TYPE ST_Robot_HMI :
STRUCT
	bStart : BOOL;
	bStop : BOOL;
	bInit : BOOL;
	bPowerOn : BOOL;
	bPowerOff : BOOL;
	
	iStep : 	UINT;
	sStatus : STRING;
END_STRUCT
END_TYPE

(* stored: Version 1.1.0.1
   DUT ST_Robot_HMI: Id {31e11358-927d-466d-8121-ae8e920930e4} *)
